(* IEC 61131-3 sources: moqui-plc/simatic-ax/src/moqui/framework/src/main/org/moqui/motion (part 2) *)

                        hasPending := FALSE;
                    END_IF;

                    commandAborted := TRUE;
                    internalStatus := AxisInternalStatus#Ready;
                ELSE
                    pendingCmd := cmd;
                    pendingOldPosition := position; pendingOldDistance := distance; pendingOldVelocity := velocity;
                    pendingOldRatioNumerator := ratioNumerator; pendingOldRatioDenominator := ratioDenominator;
                    pendingOldCamVersion := camVersion; pendingOldStartMode := startMode;
                    pendingOldMasterOffset := masterOffset; pendingOldSlaveOffset := slaveOffset;
                    hasPending := TRUE;
                    oldCmd := pendingCmd;

                    CASE pendingCmd OF
                        AxisCmd#MoveVelocity : moveVelocityExecute := TRUE;
                        AxisCmd#MoveAbsolute : moveAbsoluteExecute := TRUE;
                        AxisCmd#MoveRelative : moveRelativeExecute := TRUE;
                        AxisCmd#MoveAdditive : moveAdditiveExecute := TRUE;
                        AxisCmd#MoveSuperimposed : moveSuperimposedExecute := TRUE;
                        AxisCmd#Halt : haltExecute := TRUE;
                        AxisCmd#GearIn : gearInExecute := TRUE;
                        AxisCmd#GearInPos : gearInPosExecute := TRUE;
                        AxisCmd#CamIn : camInExecute := TRUE;
                        AxisCmd#Phasing : phasingExecute := TRUE;
                        AxisCmd#SetPosition : setPositionExecute := TRUE;
                        AxisCmd#PositionProfile : posProfileExecute := TRUE;
                        AxisCmd#VelocityProfile : velProfileExecute := TRUE;
                        AxisCmd#AccelerationProfile: accProfileExecute := TRUE;
                    ELSE
						hasPending := FALSE;
						commandAborted := TRUE;
						internalStatus := AxisInternalStatus#Ready;
                    END_CASE;
                END_IF;
            END_IF;

        (* AccelerationProfile *)
        AxisInternalStatus#AccelerationProfileState :
            IF mcAccProfile.Done THEN
                accProfileExecute := FALSE;
                IF hasPending THEN
                    hasPending := FALSE;
                    oldPosition := pendingOldPosition; oldDistance := pendingOldDistance; oldVelocity := pendingOldVelocity;
                    oldRatioNumerator := pendingOldRatioNumerator; oldRatioDenominator := pendingOldRatioDenominator;
                    oldCamVersion := pendingOldCamVersion; oldStartMode := pendingOldStartMode;
                    oldMasterOffset := pendingOldMasterOffset; oldSlaveOffset := pendingOldSlaveOffset;
                    commandExecuted := FALSE; commandAborted := FALSE;

                    CASE oldCmd OF
                        AxisCmd#MoveVelocity : internalStatus := AxisInternalStatus#MoveVelocityState;
                        AxisCmd#MoveAbsolute : internalStatus := AxisInternalStatus#MoveAbsoluteState;
                        AxisCmd#MoveRelative : internalStatus := AxisInternalStatus#MoveRelativeState;
                        AxisCmd#MoveAdditive : internalStatus := AxisInternalStatus#MoveAdditiveState;
                        AxisCmd#MoveSuperimposed : internalStatus := AxisInternalStatus#MoveSuperimposedState;
                        AxisCmd#Halt : internalStatus := AxisInternalStatus#HaltState;
                        AxisCmd#GearIn : internalStatus := AxisInternalStatus#GearInState;
                        AxisCmd#GearInPos : internalStatus := AxisInternalStatus#GearInPosState;
                        AxisCmd#CamIn : internalStatus := AxisInternalStatus#CamInState;
                        AxisCmd#Phasing : internalStatus := AxisInternalStatus#PhasingState;
                        AxisCmd#SetPosition : internalStatus := AxisInternalStatus#SetPositionState;
                        AxisCmd#PositionProfile : internalStatus := AxisInternalStatus#PositionProfileState;
                        AxisCmd#VelocityProfile : internalStatus := AxisInternalStatus#VelocityProfileState;
                        AxisCmd#AccelerationProfile: internalStatus := AxisInternalStatus#AccelerationProfileState;
                    ELSE
						internalStatus := AxisInternalStatus#Ready;
                    END_CASE;
                ELSE
                    commandExecuted := TRUE;
                    internalStatus := AxisInternalStatus#Ready;
                END_IF;
            END_IF;
            IF cmd <> oldCmd THEN
                IF bufferMode = Motion.MC_BUFFER_MODE#aborting OR hasPending THEN
                    accProfileExecute := FALSE;
                    IF hasPending THEN
                        CASE pendingCmd OF
                            AxisCmd#MoveVelocity : moveVelocityExecute := FALSE;
                            AxisCmd#MoveAbsolute : moveAbsoluteExecute := FALSE;
                            AxisCmd#MoveRelative : moveRelativeExecute := FALSE;
                            AxisCmd#MoveAdditive : moveAdditiveExecute := FALSE;
                            AxisCmd#MoveSuperimposed : moveSuperimposedExecute := FALSE;
                            AxisCmd#Halt : haltExecute := FALSE;
                            AxisCmd#GearIn : gearInExecute := FALSE;
                            AxisCmd#GearInPos : gearInPosExecute := FALSE;
                            AxisCmd#CamIn : camInExecute := FALSE;
                            AxisCmd#Phasing : phasingExecute := FALSE;
                            AxisCmd#SetPosition : setPositionExecute := FALSE;
                            AxisCmd#PositionProfile : posProfileExecute := FALSE;
                            AxisCmd#VelocityProfile : velProfileExecute := FALSE;
                            AxisCmd#AccelerationProfile: accProfileExecute := FALSE;
                        END_CASE;

                        hasPending := FALSE;
                    END_IF;

                    commandAborted := TRUE;
                    internalStatus := AxisInternalStatus#Ready;
                ELSE
                    pendingCmd := cmd;
                    pendingOldPosition := position; pendingOldDistance := distance; pendingOldVelocity := velocity;
                    pendingOldRatioNumerator := ratioNumerator; pendingOldRatioDenominator := ratioDenominator;
                    pendingOldCamVersion := camVersion; pendingOldStartMode := startMode;
                    pendingOldMasterOffset := masterOffset; pendingOldSlaveOffset := slaveOffset;
                    hasPending := TRUE;
                    oldCmd := pendingCmd;

                    CASE pendingCmd OF
                        AxisCmd#MoveVelocity : moveVelocityExecute := TRUE;
                        AxisCmd#MoveAbsolute : moveAbsoluteExecute := TRUE;
                        AxisCmd#MoveRelative : moveRelativeExecute := TRUE;
                        AxisCmd#MoveAdditive : moveAdditiveExecute := TRUE;
                        AxisCmd#MoveSuperimposed : moveSuperimposedExecute := TRUE;
                        AxisCmd#Halt : haltExecute := TRUE;
                        AxisCmd#GearIn : gearInExecute := TRUE;
                        AxisCmd#GearInPos : gearInPosExecute := TRUE;
                        AxisCmd#CamIn : camInExecute := TRUE;
                        AxisCmd#Phasing : phasingExecute := TRUE;
                        AxisCmd#SetPosition : setPositionExecute := TRUE;
                        AxisCmd#PositionProfile : posProfileExecute := TRUE;
                        AxisCmd#VelocityProfile : velProfileExecute := TRUE;
                        AxisCmd#AccelerationProfile: accProfileExecute := TRUE;
                    ELSE
						hasPending := FALSE;
						commandAborted := TRUE;
						internalStatus := AxisInternalStatus#Ready;
                    END_CASE;
                END_IF;
            END_IF;

        (* ReadParameter *)
        AxisInternalStatus#ReadParameterState :
            IF readParameter.Valid THEN
                readParameterExecute := FALSE;
                parameterReadValue := readParameter.Value;
                commandExecuted := TRUE;
                internalStatus := AxisInternalStatus#Ready;
            END_IF;
            IF cmd <> oldCmd THEN
                readParameterExecute := FALSE;
                commandAborted := TRUE;
                internalStatus := AxisInternalStatus#Ready;
            END_IF;

        (* WriteParameter *)
        AxisInternalStatus#WriteParameterState :
            IF writeParameter.Done THEN
                writeParameterExecute := FALSE;
                commandExecuted := TRUE;
                internalStatus := AxisInternalStatus#Ready;
            END_IF;
            IF cmd <> oldCmd THEN
                writeParameterExecute := FALSE;
                commandAborted := TRUE;
                internalStatus := AxisInternalStatus#Ready;
            END_IF;

        (* ReadBoolParameter *)
        AxisInternalStatus#ReadBoolParameterState :
            IF readBoolParameter.Valid THEN
                readBoolParameterExecute := FALSE;
                parameterBoolRead := readBoolParameter.Value;
                commandExecuted := TRUE;
                internalStatus := AxisInternalStatus#Ready;
            END_IF;
            IF cmd <> oldCmd THEN
                readBoolParameterExecute := FALSE;
                commandAborted := TRUE;
                internalStatus := AxisInternalStatus#Ready;
            END_IF;

        (* WriteBoolParameter *)
        AxisInternalStatus#WriteBoolParameterState :
            IF writeBoolParameter.Done THEN
                writeBoolParameterExecute := FALSE;
                commandExecuted := TRUE;
                internalStatus := AxisInternalStatus#Ready;
            END_IF;
            IF cmd <> oldCmd THEN
                writeBoolParameterExecute := FALSE;
                commandAborted := TRUE;
                internalStatus := AxisInternalStatus#Ready;
            END_IF;

        (* TouchProbe - capture axis position on hardware trigger *)
        AxisInternalStatus#TouchProbeState :
            IF touchProbe.Done THEN
                touchProbeExecute := FALSE;
                touchProbeValue := touchProbe.RecordedPosition;
                commandExecuted := TRUE;
                internalStatus := AxisInternalStatus#Ready;
            END_IF;
            IF cmd <> oldCmd THEN
                touchProbeExecute := FALSE;
                commandAborted := TRUE;
                internalStatus := AxisInternalStatus#Ready;
            END_IF;

        (* AbortTrigger - cancel any pending touch probe *)
        AxisInternalStatus#AbortTriggerState :
            IF abortTrigger.Done THEN
                abortTriggerExecute := FALSE;
                commandExecuted := TRUE;
                internalStatus := AxisInternalStatus#Ready;
            END_IF;
            IF cmd <> oldCmd THEN
                abortTriggerExecute := FALSE;
                commandAborted := TRUE;
                internalStatus := AxisInternalStatus#Ready;
            END_IF;
    END_CASE;

END_IF; (* End error-recovery guard *)

(*
 * Status Handler - level-triggered, unconditional, every cycle
 *)
readActualPosition(
    Axis := slave,
    Enable := TRUE
);
actualPosition := readActualPosition.Position;

readActualVelocity(
    Axis := slave,
    Enable := TRUE
);
actualVelocity := readActualVelocity.Velocity;

readActualTorque(
    Axis := slave,
    Enable := TRUE
);
actualTorque := readActualTorque.Torque;

readAxisError(
    Axis := slave,
    Enable := TRUE
);
axisErrorId := readAxisError.AxisErrorID;

readStatus(
    Axis := slave,
    Enable := TRUE
);
(* Priority order matches PLCopen FSM: ErrorStop > Disabled > Stopping > Homing > motion states > Standstill *)
IF readStatus.ErrorStop THEN
    status := AxisStatus#ErrorStop;
ELSIF readStatus.Disabled THEN
    status := AxisStatus#Disabled;
ELSIF readStatus.Stopping THEN
    status := AxisStatus#Stopping;
ELSIF readStatus.Homing THEN
    status := AxisStatus#Homing;
ELSIF readStatus.SynchronizedMotion THEN
    status := AxisStatus#SynchronizedMotion;
ELSIF readStatus.ContinuousMotion THEN
    status := AxisStatus#ContinuousMotion;
ELSIF readStatus.DiscreteMotion THEN
    status := AxisStatus#DiscreteMotion;
ELSIF readStatus.Standstill THEN
    status := AxisStatus#Standstill;
ELSE
    status := AxisStatus#Standstill; (* Fallback - consider adding Unknown to AxisStatus DUT *)
END_IF;

(*
 * PLCopen FB calls - unconditional every PLC cycle.
 * Execute / Enable signals are generated exclusively by the FSM above.
 * All motion parameters come directly from VAR_INPUT each cycle.
 *)

(* Administrative / Configuration *)
power(
    Axis := slave,
    Enable := powerEnable,
    bRegulatorOn := powerEnable,
    bDriveStart := powerEnable
);

resetCmd(
    Axis := slave,
    Execute := resetCmdExecute
);

setPosition(
    Axis := slave,
    Execute := setPositionExecute,
    Position := position,
    Mode := setPositionMode
);

(* Homing *)
home(
    Axis := slave,
    Execute := homeExecute,
    Position := homePosition
);

(* Motion *)
moveVelocity(
    Axis := slave,
    Execute := moveVelocityExecute,
    Velocity := velocity,
    Acceleration := acceleration,
    Deceleration := deceleration,
    Jerk := jerk,
    Direction := direction,
    BufferMode := bufferMode
);

moveAbsolute(
    Axis := slave,
    Execute := moveAbsoluteExecute,
    Position := position,
    Velocity := velocity,
    Acceleration := acceleration,
    Deceleration := deceleration,
    Jerk := jerk,
    Direction := direction,
    BufferMode := bufferMode
);

moveRelative(
    Axis := slave,
    Execute := moveRelativeExecute,
    Distance := distance,
    Velocity := velocity,
    Acceleration := acceleration,
    Deceleration := deceleration,
    Jerk := jerk,
    BufferMode := bufferMode
);

moveAdditive(
    Axis := slave,
    Execute := moveAdditiveExecute,
    Distance := distance,
    Velocity := velocity,
    Acceleration := acceleration,
    Deceleration := deceleration,
    Jerk := jerk
);

moveSuperimposed(
    Axis := slave,
    Execute := moveSuperimposedExecute,
    Distance := distance,
    VelocityDiff := velocityDiff,
    Acceleration := acceleration,
    Deceleration := deceleration,
    Jerk := jerk
);

halt(
    Axis := slave,
    Execute := haltExecute,
    Deceleration := deceleration,
    Jerk := jerk
);

haltSuperimposed(
    Axis := slave,
    Execute := haltSuperimposedExecute,
    Deceleration := deceleration,
    Jerk := jerk
);

stop(
    Axis := slave,
    Execute := stopExecute,
    Deceleration := deceleration,
    Jerk := jerk
);

jog(
    Axis := slave,
    JogForward := jogForward AND (internalStatus = AxisInternalStatus#JogState),
    JogBackward := jogBackward AND (internalStatus = AxisInternalStatus#JogState),
    Velocity := velocity,
    Acceleration := acceleration,
    Deceleration := deceleration,
    Jerk := jerk
);

(* Override *)
setOverride(
    Axis := slave,
    Enable := overrideEnable,
    VelFactor := velFactor,
    AccFactor := accFactor,
    JerkFactor := jerkFactor
);

(* Synchronization - master reference required *)
IF master <> NULL THEN
    gearIn(
        Master := master,
        Slave := slave,
        Execute := gearInExecute,
        RatioNumerator := ratioNumerator,
        RatioDenominator := TO_UDINT(ratioDenominator),
        Acceleration := acceleration,
        Deceleration := deceleration,
        Jerk := jerk,
        BufferMode := bufferMode
    );
    gearInPos(
        Master := master,
        Slave := slave,
        Execute := gearInPosExecute,
        RatioNumerator := ratioNumerator,
        RatioDenominator := ratioDenominator,
        MasterSyncPosition := masterSyncPos,
        SlaveSyncPosition := slaveSyncPos
    );
    camIn(
        Master := master,
        Slave := slave,
        Execute := camInExecute,
        CamTableID := camId,
        StartMode := startMode,
        MasterOffset := masterOffset,
        SlaveOffset := slaveOffset,
        BufferMode := bufferMode
    );
    phasing(
        Master := master,
        Slave := slave,
        Execute := phasingExecute,
        PhaseShift := phaseShift,
        Velocity := velocity,
        Acceleration := acceleration,
        Deceleration := deceleration,
        Jerk := jerk
    );
END_IF;

gearOut(
    Slave := slave,
    Execute := gearOutExecute
);

camOut(
    Slave := slave,
    Execute := camOutExecute
);

(* Profiles *)
IF positionProfile <> NULL THEN
    mcPositionProfile(
        Axis := slave,
        Execute := posProfileExecute,
        TimePosition := positionProfile
    );
END_IF;

IF velocityProfile <> NULL THEN
    mcVelocityProfile(
        Axis := slave,
        Execute := velProfileExecute,
        TimeVelocity := velocityProfile
    );
END_IF;

IF accelerationProfile <> NULL THEN
    mcAccProfile(
        Axis := slave,
        Execute := accProfileExecute,
        TimeAcceleration := accelerationProfile
    );
END_IF;

(* Parameter access *)
readParameter(
    Axis := slave,
    Enable := readParameterExecute,
    ParameterNumber := parameterNumber
);

writeParameter(
    Axis := slave,
    Execute := writeParameterExecute,
    ParameterNumber := parameterNumber,
    Value := parameterValue
);

readBoolParameter(
    Axis := slave,
    Enable := readBoolParameterExecute,
    ParameterNumber := parameterNumber
);

writeBoolParameter(
    Axis := slave,
    Execute := writeBoolParameterExecute,
    ParameterNumber := parameterNumber,
    Value := parameterBoolValue
);

(* Additional services - triggerInput reference required *)
IF triggerInput <> NULL THEN
    touchProbe(
        Axis := slave,
        Execute := touchProbeExecute,
        TriggerInput := triggerInput,
        WindowOnly := touchProbeWindow,
        FirstPosition := touchProbeFirst,
        LastPosition := touchProbeLast
    );
    abortTrigger(
        Axis := slave,
        Execute := abortTriggerExecute,
        TriggerInput := triggerInput
    );
END_IF;
END_FUNCTION_BLOCK

(* ---- AxisMotionCompat.st ---- *)
(* Compile-only compatibility stubs for Motion profile.
   Provides CODESYS Motion namespace types and MC_ function-block shells
   that Axis.st references.  No runtime logic here. *)

NAMESPACE Motion

    TYPE
        MC_BUFFER_MODE : USINT
            ( aborting      := USINT#0
            , buffered      := USINT#1
            , blendingLow   := USINT#2
            , blendingPrev  := USINT#3
            , blendingNext  := USINT#4
            , blendingHigh  := USINT#5 ) := USINT#0;

        (* IEC-61131-3 is case-insensitive: MC_Direction = MC_DIRECTION *)
        MC_Direction : USINT
            ( positive         := USINT#1
            , negative         := USINT#2
            , currentDirection := USINT#3
            , shortest         := USINT#4 ) := USINT#1;

        MC_STARTMODE : USINT
            ( absolute  := USINT#0
            , relative  := USINT#1
            , additive  := USINT#2 ) := USINT#0;

        MC_CAM_ID : STRUCT
            value : DWORD;
        END_STRUCT;

        AXIS_REF_SM3 : STRUCT
            dummy : BOOL;
        END_STRUCT;

        TRIGGER_REF : STRUCT
            dummy : BOOL;
        END_STRUCT;

        MC_TP_REF : STRUCT
            dummy : BOOL;
        END_STRUCT;

        MC_TV_REF : STRUCT
            dummy : BOOL;
        END_STRUCT;

        MC_TA_REF : STRUCT
            dummy : BOOL;
        END_STRUCT;
    END_TYPE

END_NAMESPACE

(* Axis object reference used as VAR_IN_OUT in Axis.st *)
TYPE
    TO_SynchronousAxis : STRUCT
        wDriveId : WORD;
        dummy    : BOOL;
    END_STRUCT;
END_TYPE

FUNCTION TO_STRING : STRING
VAR_INPUT
    value : WORD;
END_VAR
    TO_STRING := System.Strings.ToString(value);
END_FUNCTION

FUNCTION_BLOCK MC_Power
VAR_IN_OUT
    Axis            : TO_SynchronousAxis;
END_VAR
VAR_INPUT
    Enable          : BOOL;
    EnablePositive  : BOOL;
    EnableNegative  : BOOL;
    bRegulatorOn    : BOOL;
    bDriveStart     : BOOL;
END_VAR
VAR_OUTPUT
    Status  : BOOL;
    Busy    : BOOL;
    Error   : BOOL;
    ErrorID : DWORD;
END_VAR
END_FUNCTION_BLOCK

FUNCTION_BLOCK MC_Reset
VAR_IN_OUT
    Axis    : TO_SynchronousAxis;
END_VAR
VAR_INPUT
    Execute : BOOL;
END_VAR
VAR_OUTPUT
    Done    : BOOL;
    Busy    : BOOL;
    Error   : BOOL;
    ErrorID : DWORD;
END_VAR
END_FUNCTION_BLOCK

FUNCTION_BLOCK MC_SetPosition
VAR_IN_OUT
    Axis     : TO_SynchronousAxis;
END_VAR
VAR_INPUT
    Execute  : BOOL;
    Position : LREAL;
    Mode     : BOOL;
END_VAR
VAR_OUTPUT
    Done    : BOOL;
    Busy    : BOOL;
    Error   : BOOL;
    ErrorID : DWORD;
END_VAR
END_FUNCTION_BLOCK

FUNCTION_BLOCK MC_Home
VAR_IN_OUT
    Axis       : TO_SynchronousAxis;
END_VAR
VAR_INPUT
    Execute    : BOOL;
    Position   : LREAL;
    HomingMode : INT;
END_VAR
VAR_OUTPUT
    Done           : BOOL;
    Busy           : BOOL;
    CommandAborted : BOOL;
    Error          : BOOL;
    ErrorID        : DWORD;
END_VAR
END_FUNCTION_BLOCK

FUNCTION_BLOCK MC_MoveVelocity
VAR_IN_OUT
    Axis         : TO_SynchronousAxis;
END_VAR
VAR_INPUT
    Execute      : BOOL;
    Velocity     : REAL;
    Acceleration : REAL;
    Deceleration : REAL;
    Jerk         : REAL;
    Direction    : Motion.MC_Direction;
    BufferMode   : Motion.MC_BUFFER_MODE;
END_VAR
VAR_OUTPUT
    InVelocity     : BOOL;
    Busy           : BOOL;
    CommandAborted : BOOL;
    Error          : BOOL;
    ErrorID        : DWORD;
END_VAR
END_FUNCTION_BLOCK

FUNCTION_BLOCK MC_MoveAbsolute
VAR_IN_OUT
    Axis         : TO_SynchronousAxis;
END_VAR
VAR_INPUT
    Execute      : BOOL;
    Position     : REAL;
    Velocity     : REAL;
    Acceleration : REAL;
    Deceleration : REAL;
    Jerk         : REAL;
    Direction    : Motion.MC_Direction;
    BufferMode   : Motion.MC_BUFFER_MODE;
END_VAR
VAR_OUTPUT
    Done           : BOOL;
    Busy           : BOOL;
    CommandAborted : BOOL;
    Error          : BOOL;
    ErrorID        : DWORD;
END_VAR
END_FUNCTION_BLOCK

FUNCTION_BLOCK MC_MoveRelative
VAR_IN_OUT
    Axis         : TO_SynchronousAxis;
END_VAR
VAR_INPUT
    Execute      : BOOL;
    Distance     : REAL;
    Velocity     : REAL;
    Acceleration : REAL;
    Deceleration : REAL;
    Jerk         : REAL;
    BufferMode   : Motion.MC_BUFFER_MODE;
END_VAR
VAR_OUTPUT
    Done           : BOOL;
    Busy           : BOOL;
    CommandAborted : BOOL;
    Error          : BOOL;
    ErrorID        : DWORD;
END_VAR
END_FUNCTION_BLOCK

FUNCTION_BLOCK MC_MoveAdditive
VAR_IN_OUT
    Axis         : TO_SynchronousAxis;
END_VAR
VAR_INPUT
    Execute      : BOOL;
    Distance     : REAL;
    Velocity     : REAL;
    Acceleration : REAL;
    Deceleration : REAL;
    Jerk         : REAL;
    BufferMode   : Motion.MC_BUFFER_MODE;
END_VAR
VAR_OUTPUT
    Done           : BOOL;
    Busy           : BOOL;
    CommandAborted : BOOL;
    Error          : BOOL;
    ErrorID        : DWORD;
END_VAR
END_FUNCTION_BLOCK

FUNCTION_BLOCK MC_MoveSuperImposed
VAR_IN_OUT
    Axis             : TO_SynchronousAxis;
END_VAR
VAR_INPUT
    Execute          : BOOL;
    Distance         : REAL;
    VelocityDiff     : REAL;
    Acceleration     : REAL;
    Deceleration     : REAL;
    Jerk             : REAL;
    AccelerationDiff : REAL;
    DecelerationDiff : REAL;
    JerkDiff         : REAL;
    BufferMode       : Motion.MC_BUFFER_MODE;
END_VAR
VAR_OUTPUT
    Done           : BOOL;
    Busy           : BOOL;
    CommandAborted : BOOL;
    Error          : BOOL;
    ErrorID        : DWORD;
END_VAR
END_FUNCTION_BLOCK

FUNCTION_BLOCK MC_Halt
VAR_IN_OUT
    Axis         : TO_SynchronousAxis;
END_VAR
VAR_INPUT
    Execute      : BOOL;
    Deceleration : REAL;
    Jerk         : REAL;
    BufferMode   : Motion.MC_BUFFER_MODE;
END_VAR
VAR_OUTPUT
    Done           : BOOL;
    Busy           : BOOL;
    CommandAborted : BOOL;
    Error          : BOOL;
    ErrorID        : DWORD;
END_VAR
END_FUNCTION_BLOCK

FUNCTION_BLOCK MC_HaltSuperImposed
VAR_IN_OUT
    Axis         : TO_SynchronousAxis;
END_VAR
VAR_INPUT
    Execute      : BOOL;
    Deceleration : REAL;
    Jerk         : REAL;
END_VAR
VAR_OUTPUT
    Done           : BOOL;
    Busy           : BOOL;
    CommandAborted : BOOL;
    Error          : BOOL;
    ErrorID        : DWORD;
END_VAR
END_FUNCTION_BLOCK

FUNCTION_BLOCK MC_Stop
VAR_IN_OUT
    Axis         : TO_SynchronousAxis;
END_VAR
VAR_INPUT
    Execute      : BOOL;
    Deceleration : REAL;
    Jerk         : REAL;
END_VAR
VAR_OUTPUT
    Done    : BOOL;
    Busy    : BOOL;
    Error   : BOOL;
    ErrorID : DWORD;
END_VAR
END_FUNCTION_BLOCK

FUNCTION_BLOCK MC_Jog
VAR_IN_OUT
    Axis         : TO_SynchronousAxis;
END_VAR
VAR_INPUT
    JogForward   : BOOL;
    JogBackward  : BOOL;
    Velocity     : REAL;
    Acceleration : REAL;
    Deceleration : REAL;
    Jerk         : REAL;
END_VAR
VAR_OUTPUT
    Busy    : BOOL;
    Error   : BOOL;
    ErrorID : DWORD;
END_VAR
END_FUNCTION_BLOCK

FUNCTION_BLOCK MC_SetOverride
VAR_IN_OUT
    Axis       : TO_SynchronousAxis;
END_VAR
VAR_INPUT
    Enable     : BOOL;
    VelFactor  : REAL;
    AccFactor  : REAL;
    JerkFactor : REAL;
END_VAR
VAR_OUTPUT
    Enabled : BOOL;
    Busy    : BOOL;
    Error   : BOOL;
    ErrorID : DWORD;
END_VAR
END_FUNCTION_BLOCK

FUNCTION_BLOCK MC_GearIn
VAR_IN_OUT
    Slave            : TO_SynchronousAxis;
END_VAR
VAR_INPUT
    Master           : REF_TO Motion.AXIS_REF_SM3;
    Execute          : BOOL;
    RatioNumerator   : DINT;
    RatioDenominator : UDINT;
    Acceleration     : REAL;
    Deceleration     : REAL;
    Jerk             : REAL;
    BufferMode       : Motion.MC_BUFFER_MODE;
END_VAR
VAR_OUTPUT
    InSync         : BOOL;
    InGear         : BOOL;
    Busy           : BOOL;
    CommandAborted : BOOL;
    Error          : BOOL;
    ErrorID        : DWORD;
END_VAR
END_FUNCTION_BLOCK

FUNCTION_BLOCK MC_GearInPos
VAR_IN_OUT
    Slave               : TO_SynchronousAxis;
END_VAR
VAR_INPUT
    Master              : REF_TO Motion.AXIS_REF_SM3;
    Execute             : BOOL;
    RatioNumerator      : DINT;
    RatioDenominator    : DINT;
    MasterSyncPosition  : LREAL;
    SlaveSyncPosition   : LREAL;
    SyncMode            : USINT;
    Velocity            : REAL;
    Acceleration        : REAL;
    Deceleration        : REAL;
    Jerk                : REAL;
    BufferMode          : Motion.MC_BUFFER_MODE;
    StartMode           : Motion.MC_STARTMODE;
END_VAR
VAR_OUTPUT
    InSync         : BOOL;
    Busy           : BOOL;
    CommandAborted : BOOL;
    Error          : BOOL;
    ErrorID        : DWORD;
END_VAR
END_FUNCTION_BLOCK

FUNCTION_BLOCK MC_GearOut
VAR_IN_OUT
    Slave   : TO_SynchronousAxis;
END_VAR
VAR_INPUT
    Execute : BOOL;
END_VAR
VAR_OUTPUT
    Done    : BOOL;
    Busy    : BOOL;
    Error   : BOOL;
    ErrorID : DWORD;
END_VAR
END_FUNCTION_BLOCK

FUNCTION_BLOCK MC_CamIn
VAR_IN_OUT
    Slave              : TO_SynchronousAxis;
END_VAR
VAR_INPUT
    Master             : REF_TO Motion.AXIS_REF_SM3;
    Execute            : BOOL;
    CamTableID         : Motion.MC_CAM_ID;
    StartMode          : Motion.MC_STARTMODE;
    MasterOffset       : LREAL;
    SlaveOffset        : LREAL;
    Velocity           : REAL;
    Acceleration       : REAL;
    Deceleration       : REAL;
    Jerk               : REAL;
    BufferMode         : Motion.MC_BUFFER_MODE;
END_VAR
VAR_OUTPUT
    InSync         : BOOL;
    Busy           : BOOL;
    CommandAborted : BOOL;
    Error          : BOOL;
    ErrorID        : DWORD;
END_VAR
END_FUNCTION_BLOCK

FUNCTION_BLOCK MC_CamOut
VAR_IN_OUT
    Slave   : TO_SynchronousAxis;
END_VAR
VAR_INPUT
    Execute : BOOL;
END_VAR
VAR_OUTPUT
    Done    : BOOL;
    Busy    : BOOL;
    Error   : BOOL;
    ErrorID : DWORD;
END_VAR
END_FUNCTION_BLOCK

FUNCTION_BLOCK MC_Phasing
VAR_IN_OUT
    Slave        : TO_SynchronousAxis;
END_VAR
VAR_INPUT
    Master       : REF_TO Motion.AXIS_REF_SM3;
    Execute      : BOOL;
    PhaseShift   : LREAL;
    Velocity     : REAL;
    Acceleration : REAL;
    Deceleration : REAL;
    Jerk         : REAL;
    BufferMode   : Motion.MC_BUFFER_MODE;
END_VAR
VAR_OUTPUT
    Done           : BOOL;
    Busy           : BOOL;
    CommandAborted : BOOL;
    Error          : BOOL;
    ErrorID        : DWORD;
END_VAR
END_FUNCTION_BLOCK

FUNCTION_BLOCK MC_PositionProfile
VAR_IN_OUT
    Axis             : TO_SynchronousAxis;
END_VAR
VAR_INPUT
    Execute          : BOOL;
    TimePosition     : REF_TO Motion.MC_TP_REF;
    BufferMode       : Motion.MC_BUFFER_MODE;
END_VAR
VAR_OUTPUT
    Done           : BOOL;
    Busy           : BOOL;
    CommandAborted : BOOL;
    Error          : BOOL;
    ErrorID        : DWORD;
END_VAR
END_FUNCTION_BLOCK

FUNCTION_BLOCK MC_VelocityProfile
VAR_IN_OUT
    Axis             : TO_SynchronousAxis;
END_VAR
VAR_INPUT
    Execute          : BOOL;
    TimeVelocity     : REF_TO Motion.MC_TV_REF;
    BufferMode       : Motion.MC_BUFFER_MODE;
END_VAR
VAR_OUTPUT
    Done           : BOOL;
    Busy           : BOOL;
    CommandAborted : BOOL;
    Error          : BOOL;
    ErrorID        : DWORD;
END_VAR
END_FUNCTION_BLOCK

FUNCTION_BLOCK MC_AccelerationProfile
VAR_IN_OUT
    Axis                : TO_SynchronousAxis;
END_VAR
VAR_INPUT
    Execute             : BOOL;
    TimeAcceleration    : REF_TO Motion.MC_TA_REF;
    BufferMode          : Motion.MC_BUFFER_MODE;
END_VAR
VAR_OUTPUT
    Done           : BOOL;
    Busy           : BOOL;
    CommandAborted : BOOL;
    Error          : BOOL;
    ErrorID        : DWORD;
END_VAR
END_FUNCTION_BLOCK

FUNCTION_BLOCK MC_ReadParameter
VAR_IN_OUT
    Axis            : TO_SynchronousAxis;
END_VAR
VAR_INPUT
    Enable          : BOOL;
    ParameterNumber : WORD;
END_VAR
VAR_OUTPUT
    Valid   : BOOL;
    Busy    : BOOL;
    Error   : BOOL;
    ErrorID : DWORD;
    Value   : LREAL;
END_VAR
END_FUNCTION_BLOCK

FUNCTION_BLOCK MC_WriteParameter
VAR_IN_OUT
    Axis            : TO_SynchronousAxis;
END_VAR
VAR_INPUT
    Execute         : BOOL;
    ParameterNumber : WORD;
    Value           : LREAL;
END_VAR
VAR_OUTPUT
    Done    : BOOL;
    Busy    : BOOL;
    Error   : BOOL;
    ErrorID : DWORD;
END_VAR
END_FUNCTION_BLOCK

FUNCTION_BLOCK MC_ReadBoolParameter
VAR_IN_OUT
    Axis            : TO_SynchronousAxis;
END_VAR
VAR_INPUT
    Enable          : BOOL;
    ParameterNumber : WORD;
END_VAR
VAR_OUTPUT
    Valid   : BOOL;
    Busy    : BOOL;
    Error   : BOOL;
    ErrorID : DWORD;
    Value   : BOOL;
END_VAR
END_FUNCTION_BLOCK

FUNCTION_BLOCK MC_WriteBoolParameter
VAR_IN_OUT
    Axis            : TO_SynchronousAxis;
END_VAR
VAR_INPUT
    Execute         : BOOL;
    ParameterNumber : WORD;
    Value           : BOOL;
END_VAR
VAR_OUTPUT
    Done    : BOOL;
    Busy    : BOOL;
    Error   : BOOL;
    ErrorID : DWORD;
END_VAR
END_FUNCTION_BLOCK

FUNCTION_BLOCK MC_TouchProbe
VAR_IN_OUT
    Axis             : TO_SynchronousAxis;
END_VAR
VAR_INPUT
    Execute          : BOOL;
    TriggerInput     : REF_TO Motion.TRIGGER_REF;
    WindowOnly       : BOOL;
    FirstPosition    : LREAL;
    LastPosition     : LREAL;
END_VAR
VAR_OUTPUT
    Done             : BOOL;
    Busy             : BOOL;
    CommandAborted   : BOOL;
    Error            : BOOL;
    ErrorID          : DWORD;
    RecordedPosition : LREAL;
END_VAR
END_FUNCTION_BLOCK

FUNCTION_BLOCK MC_AbortTrigger
VAR_IN_OUT
    Axis         : TO_SynchronousAxis;
END_VAR
VAR_INPUT
    Execute      : BOOL;
    TriggerInput : REF_TO Motion.TRIGGER_REF;
END_VAR
VAR_OUTPUT
    Done    : BOOL;
    Busy    : BOOL;
    Error   : BOOL;
    ErrorID : DWORD;
END_VAR
END_FUNCTION_BLOCK

FUNCTION_BLOCK MC_ReadActualPosition
VAR_IN_OUT
    Axis   : TO_SynchronousAxis;
END_VAR
VAR_INPUT
    Enable : BOOL;
END_VAR
VAR_OUTPUT
    Valid    : BOOL;
    Busy     : BOOL;
    Error    : BOOL;
    ErrorID  : DWORD;
    Position : LREAL;
END_VAR
END_FUNCTION_BLOCK

FUNCTION_BLOCK MC_ReadActualVelocity
VAR_IN_OUT
    Axis   : TO_SynchronousAxis;
END_VAR
VAR_INPUT
    Enable : BOOL;
END_VAR
VAR_OUTPUT
    Valid    : BOOL;
    Busy     : BOOL;
    Error    : BOOL;
    ErrorID  : DWORD;
    Velocity : LREAL;
END_VAR
END_FUNCTION_BLOCK

FUNCTION_BLOCK MC_ReadActualTorque
VAR_IN_OUT
    Axis   : TO_SynchronousAxis;
END_VAR
VAR_INPUT
    Enable : BOOL;
END_VAR
VAR_OUTPUT
    Valid   : BOOL;
    Busy    : BOOL;
    Error   : BOOL;
    ErrorID : DWORD;
    Torque  : LREAL;
END_VAR
END_FUNCTION_BLOCK

FUNCTION_BLOCK MC_ReadAxisError
VAR_IN_OUT
    Axis   : TO_SynchronousAxis;
END_VAR
VAR_INPUT
    Enable : BOOL;
END_VAR
VAR_OUTPUT
    Valid       : BOOL;
    Busy        : BOOL;
    Error       : BOOL;
    ErrorID     : DWORD;
    AxisErrorID : DWORD;
END_VAR
END_FUNCTION_BLOCK

FUNCTION_BLOCK MC_ReadStatus
VAR_IN_OUT
    Axis               : TO_SynchronousAxis;
END_VAR
VAR_INPUT
    Enable             : BOOL;
END_VAR
VAR_OUTPUT
    Valid              : BOOL;
    Busy               : BOOL;
    Error              : BOOL;
    ErrorID            : DWORD;
    ErrorStop          : BOOL;
    Disabled           : BOOL;
    Stopping           : BOOL;
    Homing             : BOOL;
    Standstill         : BOOL;
    DiscreteMotion     : BOOL;
    ContinuousMotion   : BOOL;
    SynchronizedMotion : BOOL;
END_VAR
END_FUNCTION_BLOCK
